Fanuc KAREL source: ko00034.KL

-- PROVISIONAL review KL for V770-1; original PC SHA256 e1cfd46dbd7f85161ab124326f44ed052491090c60661dc9788aa8bda9ad5527
-- Incomplete behavior may be omitted. Consult companion uncertainty JSON. Do not deploy.
PROGRAM KO00034
%NOLOCKGROUP
BEGIN
  -- UNRESOLVED_PC offsets 5-12; opcodes 9D,23
  -- UNRESOLVED_PC offsets 17-66; opcodes 27,27,49,7E,AD,22,1C,22,31,7E,4A
  -- UNRESOLVED_PC offsets 71-75; opcodes 7F
END KO00034
